SUBAPPLICATION RequestOrchestrationOpcUaPartial (* Request Orchestration using OPC UA with all fields from services to be set *)
  (* Standard: 61499-2; Description: Copyright (c) 2019 fortiss GmbH This program and the accompanying materials are made available under the terms of the Eclipse Public License 2.0 which is available at https://www.eclipse.org/legal/epl-2.0/ SPDX-License-Identifier: EPL-2.0 *)
  (* Version 1.0, 2019-09-17, Jose Cabral, fortiss GmbH *)
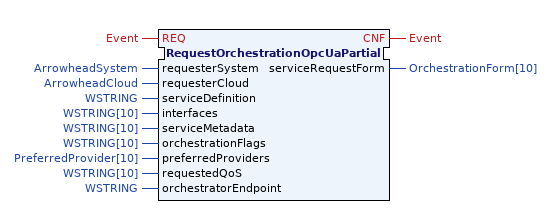
  EVENT_INPUT
    REQ; (* Request orchestration *)
  END_EVENT
  EVENT_OUTPUT
    CNF; (* Request finished *)
  END_EVENT
  VAR_INPUT
    requesterSystem : ArrowheadSystem; (* The ArrowheadSystem identifier that is requesting the orchestration *)
    requesterCloud : ArrowheadCloud; (* Not to be used by Application Systems. This field is only used when there is an inbound request from another Cloud. This can only be submitted by the Gatekeeper *)
    serviceDefinition : WSTRING; (* Identification of the service *)
    interfaces : ARRAY [0..9] OF WSTRING; (* Interfaces implemented by the service *)
    serviceMetadata : ARRAY [0..9] OF WSTRING; (* Metadata of the service in key=value format *)
    orchestrationFlags : ARRAY [0..9] OF WSTRING; (* These flags can be set to tailor the orchestration process (use just the names of the flags to be enabled) *)
    preferredProviders : ARRAY [0..9] OF PreferredProvider; (* There can be a list from the Consumer stating which other Application Systems (even from other Clouds) it wishes to connect. If this field is filled out, the Orchestrator will try to facilitate these preferences *)
    requestedQoS : ARRAY [0..9] OF WSTRING; (* This object will be presenting the Consumer’s selected QoS level. Not implemented *)
    orchestratorEndpoint : WSTRING; (* Enpoint of the orchestrator *)
  END_VAR
  VAR_OUTPUT
    serviceRequestForm : ARRAY [0..9] OF OrchestrationForm; (* Response from the orchestrator *)
  END_VAR
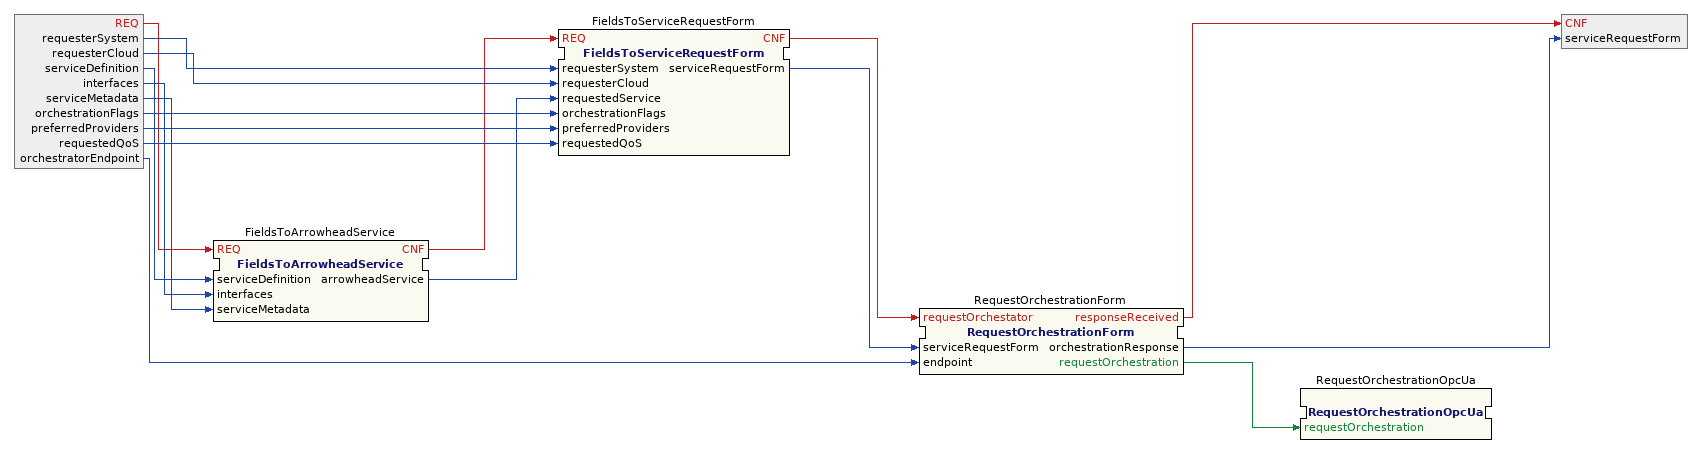
  FBS
    FieldsToServiceRequestForm : FieldsToServiceRequestForm;
    FieldsToArrowheadService : FieldsToArrowheadService;
    RequestOrchestrationForm : RequestOrchestrationForm;
    RequestOrchestrationOpcUa : RequestOrchestrationOpcUa;
  END_FBS
  EVENT_CONNECTIONS
    REQ TO FieldsToArrowheadService.REQ;
    FieldsToArrowheadService.CNF TO FieldsToServiceRequestForm.REQ;
    FieldsToServiceRequestForm.CNF TO RequestOrchestrationForm.requestOrchestator;
    RequestOrchestrationForm.responseReceived TO CNF;
  END_CONNECTIONS
  DATA_CONNECTIONS
    requesterSystem TO FieldsToServiceRequestForm.requesterSystem;
    requesterCloud TO FieldsToServiceRequestForm.requesterCloud;
    FieldsToArrowheadService.arrowheadService TO FieldsToServiceRequestForm.requestedService;
    serviceDefinition TO FieldsToArrowheadService.serviceDefinition;
    interfaces TO FieldsToArrowheadService.interfaces;
    serviceMetadata TO FieldsToArrowheadService.serviceMetadata;
    orchestrationFlags TO FieldsToServiceRequestForm.orchestrationFlags;
    preferredProviders TO FieldsToServiceRequestForm.preferredProviders;
    requestedQoS TO FieldsToServiceRequestForm.requestedQoS;
    FieldsToServiceRequestForm.serviceRequestForm TO RequestOrchestrationForm.serviceRequestForm;
    RequestOrchestrationForm.orchestrationResponse TO serviceRequestForm;
    orchestratorEndpoint TO RequestOrchestrationForm.endpoint;
  END_CONNECTIONS
  ADAPTER_CONNECTIONS
    RequestOrchestrationForm.requestOrchestration TO RequestOrchestrationOpcUa.requestOrchestration;
  END_CONNECTIONS
END_SUBAPPLICATION
